Fanuc TP program (LS listing): MOVEHOME.LS

/PROG  MOVEHOME
/ATTR
OWNER		= MNEDITOR;
COMMENT		= "macro home pt";
PROG_SIZE	= 279;
CREATE		= DATE 19-09-30  TIME 15:29:52;
MODIFIED	= DATE 19-09-30  TIME 17:36:32;
FILE_NAME	= PROGRAM_;
VERSION		= 0;
LINE_COUNT	= 4;
MEMORY_SIZE	= 635;
PROTECT		= READ_WRITE;
TCD:  STACK_SIZE	= 0,
      TASK_PRIORITY	= 50,
      TIME_SLICE	= 0,
      BUSY_LAMP_OFF	= 0,
      ABORT_REQUEST	= 0,
      PAUSE_REQUEST	= 0;
DEFAULT_GROUP	= 1,*,*,*,*;
CONTROL_CODE	= 00000000 00000000;
/APPL
/APPL

AUTO_SINGULARITY_HEADER;
  ENABLE_SINGULARITY_AVOIDANCE   : TRUE;
/MN
   1:  !Set UT & UF ;
   2:  UTOOL_NUM=1 ;
   3:  UFRAME_NUM=1 ;
   4:J PR[8:RobotHome] 100% FINE    ;
/POS
/END
